SUBAPPLICATION ErsteAutomatisierung (* Motor Links/Rechtslauf *)
  (* Standard: 61499-2; Description: Copyright (c) 2023 Meisterschulen am Ostbahnhof This program and the accompanying materials are made available under the terms of the Eclipse Public License 2.0 which is available at https://www.eclipse.org/legal/epl-2.0/ SPDX-License-Identifier: EPL-2.0 *)
  (* Version 1.0, 2023-10-23, Franz Höpfinger, Meisterschulen am Ostbahnhof, initial API and implementation and/or initial documentation *)
  PACKAGE Uebungen;
  IMPORT logiBUS::io::DI::logiBUS_DI::Input_I1;
  IMPORT logiBUS::io::DI::logiBUS_DI::Input_I2;
  IMPORT logiBUS::io::DI::logiBUS_DI::Input_I3;
  IMPORT logiBUS::io::DI::logiBUS_DI_Events::BUTTON_PRESS_DOWN;
  IMPORT logiBUS::io::DI::logiBUS_DI_Events::BUTTON_SINGLE_CLICK;
  IMPORT logiBUS::io::DQ::logiBUS_DO::Output_Q5;
  IMPORT logiBUS::io::DQ::logiBUS_DO::Output_Q56;
  IMPORT logiBUS::io::DQ::logiBUS_DO::Output_Q6;
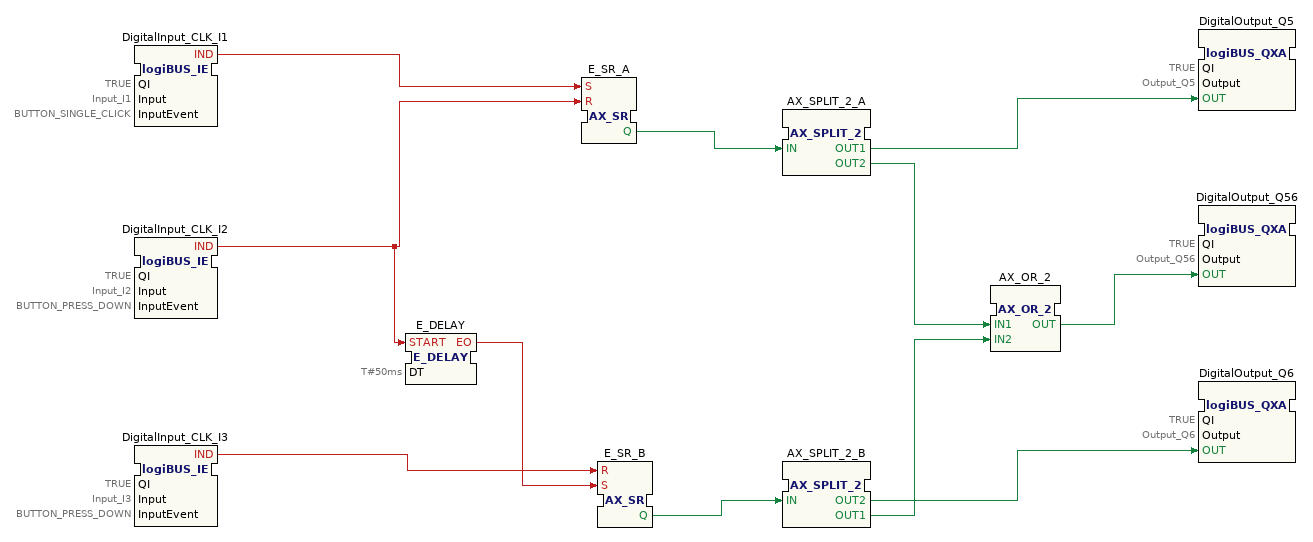
  FBS
    DigitalOutput_Q5 : logiBUS::io::DQ::logiBUS_QXA(QI := TRUE, Output := Output_Q5);
    DigitalOutput_Q6 : logiBUS::io::DQ::logiBUS_QXA(QI := TRUE, Output := Output_Q6);
    AX_OR_2 : adapter::booleanOperators::AX_OR_2;
    DigitalOutput_Q56 : logiBUS::io::DQ::logiBUS_QXA(QI := TRUE, Output := Output_Q56);
    AX_SPLIT_2_A : adapter::events::unidirectional::AX_SPLIT_2;
    AX_SPLIT_2_B : adapter::events::unidirectional::AX_SPLIT_2;
    DigitalInput_CLK_I1 : logiBUS::io::DI::logiBUS_IE(QI := TRUE, Input := Input_I1, InputEvent := BUTTON_SINGLE_CLICK);
    E_SR_A : adapter::events::unidirectional::AX_SR;
    DigitalInput_CLK_I2 : logiBUS::io::DI::logiBUS_IE(QI := TRUE, Input := Input_I2, InputEvent := BUTTON_PRESS_DOWN);
    DigitalInput_CLK_I3 : logiBUS::io::DI::logiBUS_IE(QI := TRUE, Input := Input_I3, InputEvent := BUTTON_PRESS_DOWN);
    E_SR_B : adapter::events::unidirectional::AX_SR;
    E_DELAY : iec61499::events::E_DELAY(DT := T#50ms);
  END_FBS
  EVENT_CONNECTIONS
    DigitalInput_CLK_I1.IND TO E_SR_A.S;
    DigitalInput_CLK_I2.IND TO E_SR_A.R;
    DigitalInput_CLK_I2.IND TO E_DELAY.START;
    DigitalInput_CLK_I3.IND TO E_SR_B.R;
    E_DELAY.EO TO E_SR_B.S;
  END_CONNECTIONS
  ADAPTER_CONNECTIONS
    AX_SPLIT_2_A.OUT1 TO DigitalOutput_Q5.OUT;
    AX_SPLIT_2_B.OUT2 TO DigitalOutput_Q6.OUT;
    AX_OR_2.OUT TO DigitalOutput_Q56.OUT;
    AX_SPLIT_2_A.OUT2 TO AX_OR_2.IN1;
    AX_SPLIT_2_B.OUT1 TO AX_OR_2.IN2;
    E_SR_A.Q TO AX_SPLIT_2_A.IN;
    E_SR_B.Q TO AX_SPLIT_2_B.IN;
  END_CONNECTIONS
END_SUBAPPLICATION
